TYPE ST_DB_STOFFWERTE :
STRUCT
	id: DINT;
	temp: STRING(45);
	dichte: STRING(45);
	cp: STRING(45);
END_STRUCT
END_TYPE

(* stored: Version 1.1.0.1, ProductVersion 3.1.4018.5
   DUT ST_DB_STOFFWERTE: Id {df2a5b8a-4413-49fa-899b-27aa6d251e96} *)
